INTERFACE IListItem

PROPERTY data : INT
GET
END_GET
SET
END_SET
END_PROPERTY

PROPERTY next : POINTER TO Node
GET
END_GET
SET
END_SET
END_PROPERTY

END_INTERFACE

(* stored: Version 1.1.0.1, ProductVersion 3.1.4024.11
   Itf IListItem: Id {91690c9e-d3ca-4e14-9e0a-1b3f1b6401df}
   Property data: Id {76126edc-0a12-45ac-9898-53e76a7592e2}
   Get Get: Id {2d1b33ee-bffa-43de-982f-280c66a966a5}
   Set Set: Id {6b8afa56-b726-4fe3-83d1-6fe27fa8eb5f}
   Property next: Id {26a8b14b-5e8f-4c24-949a-bbd455456cda}
   Get Get: Id {82abfbf1-bced-41fc-8a56-24bc96d84b21}
   Set Set: Id {10feaf45-ca62-4397-a278-e797045eb76b} *)
